// TIA Portal V16 export
// export: Created 2024-04-26T21:24:43.6379143Z, ExportSetting WithDefaults, DisplayName Totally Integrated Automation Portal, DisplayVersion V16, DisplayName TIA Portal Version Control Interface, DisplayVersion V16, DisplayName TIA Portal Openness, DisplayVersion V16, DisplayName STEP 7 Professional, DisplayVersion V16, DisplayName STEP 7 Safety, DisplayVersion V16, DisplayName WinCC Professional, DisplayVersion V16
DATA_BLOCK "MC_Power_DB_2"   // DB21
// stored: AutoNumber true, InstanceOfName MC_Power, OfSystemLibElement MC_Power, OfSystemLibVersion 6.0
"MC_Power"
   // VAR_INPUT
   //    Axis : TO_Axis;
   //    Enable : Bool;
   //    StartMode : Int;
   //    StopMode : Int;
   // END_VAR
   // VAR_OUTPUT
   //    Status : Bool;
   //    Busy : Bool;
   //    Error : Bool;
   //    ErrorID : Word;
   //    ErrorInfo : Word;
   // END_VAR
   // VAR
   //    FB_ID : DInt;
   // END_VAR
BEGIN
END_DATA_BLOCK
